// TIA Portal V20 export
DATA_BLOCK "InstPlcDiag"   // DB34
AUTHOR : Siemens Digital Industries
FAMILY : LAF
// stored: InstanceOfName LAF_PlcDiag, InstanceOfType FB
"LAF_PlcDiag"
   // VAR_INPUT
   //    localCommon { ExternalAccessible := 'False'; ExternalVisible := 'False'; ExternalWritable := 'False'} : HW_SUBMODULE;
   //    localProfinetInterface { ExternalAccessible := 'False'; ExternalVisible := 'False'; ExternalWritable := 'False'} : HW_INTERFACE;
   //    firstCycle { ExternalAccessible := 'False'; ExternalVisible := 'False'; ExternalWritable := 'False'} : Bool;
   // END_VAR
   // VAR_IN_OUT
   //    diagDataHmi : "LAF_typePlcDiag";
   // END_VAR
   // VAR
   //    statLocalCommon { ExternalAccessible := 'False'; ExternalVisible := 'False'; ExternalWritable := 'False'} : HW_SUBMODULE;
   //    statLocProfinetInterface { ExternalAccessible := 'False'; ExternalVisible := 'False'; ExternalWritable := 'False'} : HW_INTERFACE;
   //    instGetImData0 { ExternalAccessible := 'False'; ExternalVisible := 'False'; ExternalWritable := 'False'} : Get_IM_Data;
   //    statGetImData0ErrorSaved { ExternalAccessible := 'False'; ExternalVisible := 'False'; ExternalWritable := 'False'} : Word;
   //    instGetImData1 { ExternalAccessible := 'False'; ExternalVisible := 'False'; ExternalWritable := 'False'} : Get_IM_Data;
   //    statGetImData1ErrorSaved { ExternalAccessible := 'False'; ExternalVisible := 'False'; ExternalWritable := 'False'} : Word;
   //    instGetImData2 { ExternalAccessible := 'False'; ExternalVisible := 'False'; ExternalWritable := 'False'} : Get_IM_Data;
   //    statGetImData2ErrorSaved { ExternalAccessible := 'False'; ExternalVisible := 'False'; ExternalWritable := 'False'} : Word;
   //    instGetImData3 { ExternalAccessible := 'False'; ExternalVisible := 'False'; ExternalWritable := 'False'} : Get_IM_Data;
   //    statGetImData3ErroSaved { ExternalAccessible := 'False'; ExternalVisible := 'False'; ExternalWritable := 'False'} : Word;
   //    instReadRecord { ExternalAccessible := 'False'; ExternalVisible := 'False'; ExternalWritable := 'False'} : RDREC;
   //    statReadRecordResult { ExternalAccessible := 'False'; ExternalVisible := 'False'; ExternalWritable := 'False'} : Array[0..199] of Byte;
   //    statStartNetAddresses { ExternalAccessible := 'False'; ExternalVisible := 'False'; ExternalWritable := 'False'} : USInt;
   //    statIm1PlDesiLocIdLen { ExternalAccessible := 'False'; ExternalVisible := 'False'; ExternalWritable := 'False'} : Int;
   //    statRisEdgeReadAll { ExternalAccessible := 'False'; ExternalVisible := 'False'; ExternalWritable := 'False'} : Bool;
   //    statPosPulseReadAll { ExternalAccessible := 'False'; ExternalVisible := 'False'; ExternalWritable := 'False'} : Bool;
   //    statErrorText { ExternalAccessible := 'False'; ExternalVisible := 'False'; ExternalWritable := 'False'} : String[30];
   // END_VAR
BEGIN
END_DATA_BLOCK
